{attribute addProperty BoxType "EP2816-0008-0016"}
{attribute addProperty Id "Safe_state_activeAT %I*BOOL811Error_channelAT %I*ARRAY[0 ..1] OF BOOL1620Sync_ErrorAT %I*BOOL8132TxPDO_ToggleAT %I*BOOL819"}
{attribute addProperty CRC "493053222"}
{attribute addProperty SizeInBites "40"}
{attribute addProperty SizeInBytes "5"}
TYPE DO_Inputs_Device_213DCE55 :
STRUCT
	{attribute addProperty Name "Safe_state_active"}
	Safe_state_active AT %I* : BOOL;
	{attribute addProperty Name "Error_channel"}
	Error_channel AT %I* : ARRAY[0 ..1] OF BOOL;
	{attribute addProperty Name "Sync_Error"}
	Sync_Error AT %I* : BOOL;
	{attribute addProperty Name "TxPDO_Toggle"}
	TxPDO_Toggle AT %I* : BOOL;
END_STRUCT
END_TYPE

(* stored: Version 1.2.0.0, ProductVersion 3.1.4024.9
   DUT DO_Inputs_Device_213DCE55: Id {f4e675d8-57b5-4a50-af9f-5f3d9d5ed61b} *)
